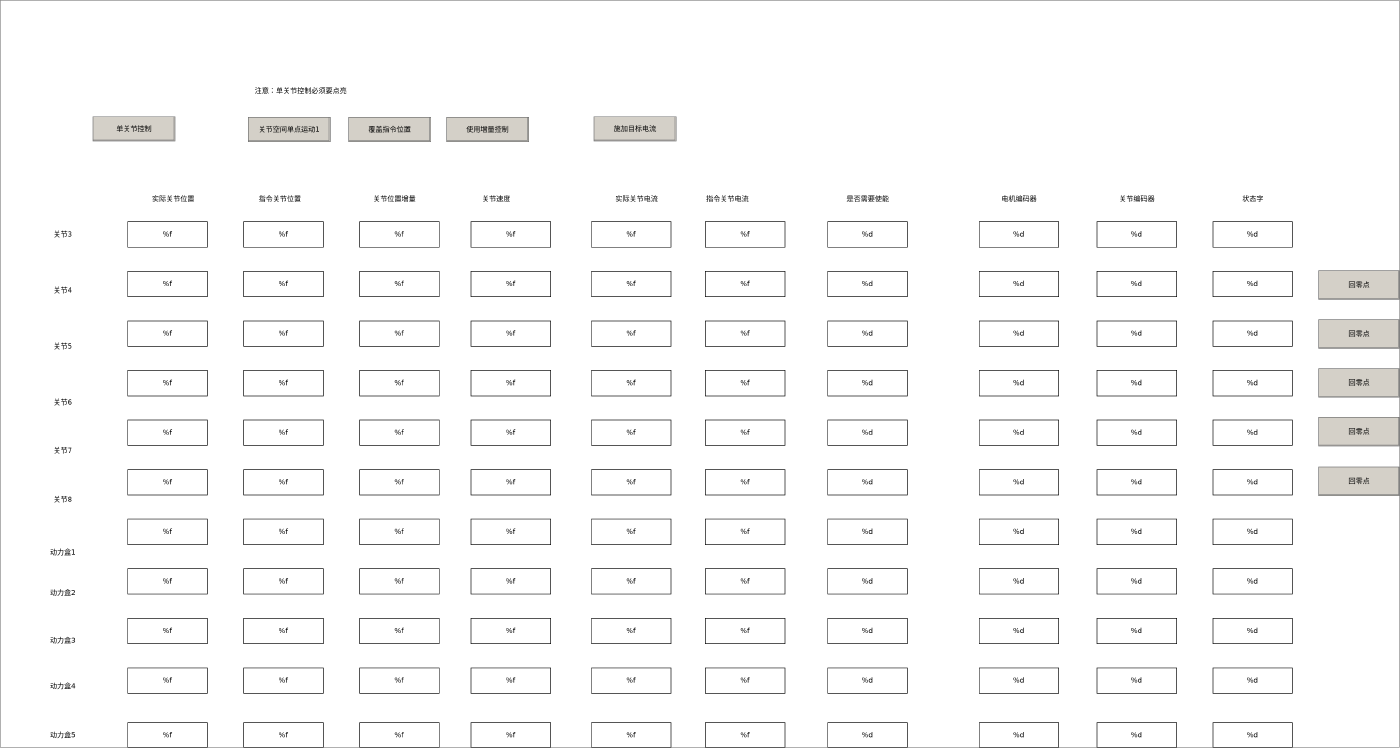
VISUALIZATION motion_a4  // 2174x1162
    Button (385,182 128x38), "关节空间单点运动1", colour toggle: g_motionTest.m_uiArmMode[4,1]
        tap g_motionTest.m_uiArmMode[1,1]
    Label (362,295 145x28), "指令关节位置"
    Label (194,294 150x30), "实际关节位置"
    Label (540,295 145x28), "关节位置增量"
    Label (698,295 145x28), "关节速度"
    Label (916,295 145x28), "实际关节电流"
    Label (1057,295 145x28), "指令关节电流"
    Rectangle (198,575 124x40), "%f", text variable: g_motionTest.m_actJntPos[4][1]
    Label (25,350 145x28), "关节3"
    Label (25,437 145x28), "关节4"
    Label (25,524 145x28), "关节5"
    Label (25,611 145x28), "关节6"
    Label (25,686 145x28), "关节7"
    Label (25,762 145x28), "关节8"
    Label (25,844 145x28), "动力盒1"
    Label (25,907 145x28), "动力盒2"
    Label (25,1128 145x28), "动力盒5"
    Label (25,981 145x28), "动力盒3"
    Label (25,1052 145x28), "动力盒4"
    Rectangle (198,652 124x40), "%f", text variable: g_motionTest.m_actJntPos[4][2]
    Rectangle (198,729 124x40), "%f", text variable: g_motionTest.m_actJntPos[4][3]
    Rectangle (198,806 124x40), "%f", text variable: g_motionTest.m_actJntPos[4][4]
    Rectangle (198,883 124x40), "%f", text variable: g_motionTest.m_actJntPos[4][5]
    Rectangle (198,960 124x40), "%f", text variable: g_motionTest.m_actJntPos[4][6]
    Rectangle (198,1037 124x40), "%f", text variable: g_motionTest.m_actJntPos[4][7]
    Rectangle (198,1122 124x40), "%f", text variable: g_motionTest.m_actJntPos[4][8]
    Rectangle (198,344 124x40), "%f", text variable: g_motionTest.m_actJntPosSetup[4][3]
    Rectangle (198,421 124x40), "%f", text variable: g_motionTest.m_actJntPosSetup[4][4]
    Rectangle (198,498 124x40), "%f", text variable: g_motionTest.m_actJntPosSetup[4][5]
    Rectangle (378,344 124x40), "%f", text variable: g_motionTest.m_targetJntPosSetup[4][3]
        OnMouseClick: write the text variable via Default
    Rectangle (378,421 124x40), "%f", text variable: g_motionTest.m_targetJntPosSetup[4][4]
        OnMouseClick: write the text variable via Default
    Rectangle (378,498 124x40), "%f", text variable: g_motionTest.m_targetJntPosSetup[4][5]
        OnMouseClick: write the text variable via Default
    Rectangle (378,575 124x40), "%f", text variable: g_motionTest.m_targetJntPosN8[4][1]
        OnMouseClick: write the text variable via Default
    Rectangle (378,652 124x40), "%f", text variable: g_motionTest.m_targetJntPosN8[4][2]
        OnMouseClick: write the text variable via Default
    Rectangle (378,729 124x40), "%f", text variable: g_motionTest.m_targetJntPosN8[4][3]
        OnMouseClick: write the text variable via Default
    Rectangle (378,806 124x40), "%f", text variable: g_motionTest.m_targetJntPosN8[4][4]
        OnMouseClick: write the text variable via Default
    Rectangle (378,883 124x40), "%f", text variable: g_motionTest.m_targetJntPosN8[4][5]
        OnMouseClick: write the text variable via Default
    Rectangle (378,960 124x40), "%f", text variable: g_motionTest.m_targetJntPosN8[4][6]
        OnMouseClick: write the text variable via Default
    Rectangle (378,1037 124x40), "%f", text variable: g_motionTest.m_targetJntPosN8[4][7]
        OnMouseClick: write the text variable via Default
    Rectangle (378,1122 124x40), "%f", text variable: g_motionTest.m_targetJntPosN8[4][8]
        OnMouseClick: write the text variable via Default
    Rectangle (558,344 124x40), "%f", text variable: g_motionTest.m_targetJntPosIncSetup[4][3]
        OnMouseClick: write the text variable via Default
    Rectangle (558,421 124x40), "%f", text variable: g_motionTest.m_targetJntPosIncSetup[4][4]
        OnMouseClick: write the text variable via Default
    Rectangle (558,498 124x40), "%f", text variable: g_motionTest.m_targetJntPosIncSetup[4][5]
        OnMouseClick: write the text variable via Default
    Rectangle (558,575 124x40), "%f", text variable: g_motionTest.m_targetJntPosIncN8[4][1]
        OnMouseClick: write the text variable via Default
    Rectangle (558,652 124x40), "%f", text variable: g_motionTest.m_targetJntPosIncN8[4][2]
        OnMouseClick: write the text variable via Default
    Rectangle (558,729 124x40), "%f", text variable: g_motionTest.m_targetJntPosIncN8[4][3]
        OnMouseClick: write the text variable via Default
    Rectangle (558,806 124x40), "%f", text variable: g_motionTest.m_targetJntPosIncN8[4][4]
        OnMouseClick: write the text variable via Default
    Rectangle (558,883 124x40), "%f", text variable: g_motionTest.m_targetJntPosIncN8[4][5]
        OnMouseClick: write the text variable via Default
    Rectangle (558,960 124x40), "%f", text variable: g_motionTest.m_targetJntPosIncN8[4][6]
        OnMouseClick: write the text variable via Default
    Rectangle (558,1037 124x40), "%f", text variable: g_motionTest.m_targetJntPosIncN8[4][7]
        OnMouseClick: write the text variable via Default
    Rectangle (558,1122 124x40), "%f", text variable: g_motionTest.m_targetJntPosIncN8[4][8]
        OnMouseClick: write the text variable via Default
    Rectangle (731,344 124x40), "%f", text variable: g_motionTest.m_targetJntVelSetup[4][3]
        OnMouseClick: write the text variable via Default
    Rectangle (731,421 124x40), "%f", text variable: g_motionTest.m_targetJntVelSetup[4][4]
        OnMouseClick: write the text variable via Default
    Rectangle (731,498 124x40), "%f", text variable: g_motionTest.m_targetJntVelSetup[4][5]
        OnMouseClick: write the text variable via Default
    Rectangle (731,575 124x40), "%f", text variable: g_motionTest.m_targetJntVel[4][1]
        OnMouseClick: write the text variable via Default
    Rectangle (731,652 124x40), "%f", text variable: g_motionTest.m_targetJntVel[4][2]
        OnMouseClick: write the text variable via Default
    Rectangle (731,729 124x40), "%f", text variable: g_motionTest.m_targetJntVel[4][3]
        OnMouseClick: write the text variable via Default
    Rectangle (731,806 124x40), "%f", text variable: g_motionTest.m_targetJntVel[4][4]
        OnMouseClick: write the text variable via Default
    Rectangle (731,883 124x40), "%f", text variable: g_motionTest.m_targetJntVel[4][5]
        OnMouseClick: write the text variable via Default
    Rectangle (731,960 124x40), "%f", text variable: g_motionTest.m_targetJntVel[4][6]
        OnMouseClick: write the text variable via Default
    Rectangle (731,1037 124x40), "%f", text variable: g_motionTest.m_targetJntVel[4][7]
        OnMouseClick: write the text variable via Default
    Rectangle (731,1122 124x40), "%f", text variable: g_motionTest.m_targetJntVel[4][8]
        OnMouseClick: write the text variable via Default
    Rectangle (918,344 124x40), "%f", text variable: g_motionTest.m_actJntCurrentSetup[4][3]
    Rectangle (918,421 124x40), "%f", text variable: g_motionTest.m_actJntCurrentSetup[4][4]
    Rectangle (918,498 124x40), "%f", text variable: g_motionTest.m_actJntCurrentSetup[4][5]
    Rectangle (918,575 124x40), "%f", text variable: g_motionTest.m_actJntCurrent[4][1]
    Rectangle (918,652 124x40), "%f", text variable: g_motionTest.m_actJntCurrent[4][2]
    Rectangle (918,729 124x40), "%f", text variable: g_motionTest.m_actJntCurrent[4][3]
    Rectangle (918,806 124x40), "%f", text variable: g_motionTest.m_actJntCurrent[4][4]
    Rectangle (918,883 124x40), "%f", text variable: g_motionTest.m_actJntCurrent[4][5]
    Rectangle (918,960 124x40), "%f", text variable: g_motionTest.m_actJntCurrent[4][6]
    Rectangle (918,1037 124x40), "%f", text variable: g_motionTest.m_actJntCurrent[4][7]
    Rectangle (918,1122 124x40), "%f", text variable: g_motionTest.m_actJntCurrent[4][8]
    Rectangle (1095,344 124x40), "%f", text variable: g_motionTest.m_targetJntCurrentSetup[4][3]
        OnMouseClick: write the text variable via Default
    Rectangle (1095,421 124x40), "%f", text variable: g_motionTest.m_targetJntCurrentSetup[4][4]
        OnMouseClick: write the text variable via Default
    Rectangle (1095,498 124x40), "%f", text variable: g_motionTest.m_targetJntCurrentSetup[4][5]
        OnMouseClick: write the text variable via Default
    Rectangle (1095,575 124x40), "%f", text variable: g_motionTest.m_targetJntCurrentN8[4][1]
        OnMouseClick: write the text variable via Default
    Rectangle (1095,652 124x40), "%f", text variable: g_motionTest.m_targetJntCurrentN8[4][2]
        OnMouseClick: write the text variable via Default
    Rectangle (1095,729 124x40), "%f", text variable: g_motionTest.m_targetJntCurrentN8[4][3]
        OnMouseClick: write the text variable via Default
    Rectangle (1095,806 124x40), "%f", text variable: g_motionTest.m_targetJntCurrentN8[4][4]
        OnMouseClick: write the text variable via Default
    Rectangle (1095,883 124x40), "%f", text variable: g_motionTest.m_targetJntCurrentN8[4][5]
        OnMouseClick: write the text variable via Default
    Rectangle (1095,960 124x40), "%f", text variable: g_motionTest.m_targetJntCurrentN8[4][6]
        OnMouseClick: write the text variable via Default
    Rectangle (1095,1037 124x40), "%f", text variable: g_motionTest.m_targetJntCurrentN8[4][7]
        OnMouseClick: write the text variable via Default
    Rectangle (1095,1122 124x40), "%f", text variable: g_motionTest.m_targetJntCurrentN8[4][8]
        OnMouseClick: write the text variable via Default
    Button (693,182 128x38), "使用增量控制", colour toggle: g_motionTest.m_singleMotorIncControl[4]
        toggle g_motionTest.m_singleMotorIncControl[4]
    Button (922,181 128x38), "施加目标电流", colour toggle: g_motionTest.m_uiArmMode[4,9]
        toggle g_motionTest.m_uiArmMode[4,9]
    Button (144,181 128x38), "单关节控制", colour toggle: g_motionTest.m_singleMotorControl[4]
        toggle g_motionTest.m_singleMotorControl[4]
    Label (357,126 220x30), "注意：单关节控制必须要点亮"
    Label (1275,294 145x30), "是否需要使能"
    Rectangle (1285,344 124x40), "%d", text variable: g_motionTest.m_jntEnableSetup[4][3]
        OnMouseClick: write the text variable via Default
    Rectangle (1285,421 124x40), "%d", text variable: g_motionTest.m_jntEnableSetup[4][4]
        OnMouseClick: write the text variable via Default
    Rectangle (1285,498 124x40), "%d", text variable: g_motionTest.m_jntEnableSetup[4][5]
        OnMouseClick: write the text variable via Default
    Rectangle (1285,575 124x40), "%d", text variable: g_motionTest.m_jntEnable[4][1]
        OnMouseClick: write the text variable via Default
    Rectangle (1285,652 124x40), "%d", text variable: g_motionTest.m_jntEnable[4][2]
        OnMouseClick: write the text variable via Default
    Label (1510,295 145x28), "电机编码器"
    Label (1693,295 145x28), "关节编码器"
    Label (1873,295 145x28), "状态字"
    Rectangle (1520,344 124x40), "%d", text variable: g_systemInfo.m_setupJntInfo[4,3].m_motorInput.m_motorEncoder
    Rectangle (1520,421 124x40), "%d", text variable: g_systemInfo.m_setupJntInfo[4,4].m_motorInput.m_motorEncoder
    Rectangle (1520,498 124x40), "%d", text variable: g_systemInfo.m_setupJntInfo[4,5].m_motorInput.m_motorEncoder
    Rectangle (1520,575 124x40), "%d", text variable: g_systemInfo.m_slaveJntInfo[4,1].m_motorInput.m_motorEncoder
    Rectangle (1520,652 124x40), "%d", text variable: g_systemInfo.m_slaveJntInfo[4,2].m_motorInput.m_motorEncoder
    Rectangle (1703,344 124x40), "%d", text variable: g_systemInfo.m_setupJntInfo[4,3].m_motorInput.m_linkEncoder
    Rectangle (1703,421 124x40), "%d", text variable: g_systemInfo.m_setupJntInfo[4,4].m_motorInput.m_linkEncoder
    Rectangle (1703,498 124x40), "%d", text variable: g_systemInfo.m_setupJntInfo[4,5].m_motorInput.m_linkEncoder
    Rectangle (1703,575 124x40), "%d", text variable: g_systemInfo.m_slaveJntInfo[4,1].m_motorInput.m_linkEncoder
    Rectangle (1703,652 124x40), "%d", text variable: g_systemInfo.m_slaveJntInfo[4,2].m_motorInput.m_linkEncoder
    Rectangle (1883,344 124x40), "%d", text variable: g_systemInfo.m_setupJntInfo[4,3].m_motorInput.m_statusWord
    Rectangle (1883,421 124x40), "%d", text variable: g_systemInfo.m_setupJntInfo[4,4].m_motorInput.m_statusWord
    Rectangle (1883,498 124x40), "%d", text variable: g_systemInfo.m_setupJntInfo[4,5].m_motorInput.m_statusWord
    Rectangle (1883,575 124x40), "%d", text variable: g_systemInfo.m_slaveJntInfo[4,1].m_motorInput.m_statusWord
    Rectangle (1883,652 124x40), "%d", text variable: g_systemInfo.m_slaveJntInfo[4,2].m_motorInput.m_statusWord
    Rectangle (1520,729 124x40), "%d", text variable: g_systemInfo.m_slaveJntInfo[4,3].m_motorInput.m_motorEncoder
    Rectangle (1520,806 124x40), "%d", text variable: g_systemInfo.m_slaveJntInfo[4,4].m_motorInput.m_motorEncoder
    Rectangle (1520,883 124x40), "%d", text variable: g_systemInfo.m_slaveJntInfo[4,5].m_motorInput.m_motorEncoder
    Rectangle (1520,960 124x40), "%d", text variable: g_systemInfo.m_slaveJntInfo[4,6].m_motorInput.m_motorEncoder
    Rectangle (1520,1037 124x40), "%d", text variable: g_systemInfo.m_slaveJntInfo[4,7].m_motorInput.m_motorEncoder
    Rectangle (1520,1122 124x40), "%d", text variable: g_systemInfo.m_slaveJntInfo[4,8].m_motorInput.m_motorEncoder
    Rectangle (1703,729 124x40), "%d", text variable: g_systemInfo.m_slaveJntInfo[4,3].m_motorInput.m_linkEncoder
    Rectangle (1703,806 124x40), "%d", text variable: g_systemInfo.m_slaveJntInfo[4,4].m_motorInput.m_linkEncoder
    Rectangle (1703,883 124x40), "%d", text variable: g_systemInfo.m_slaveJntInfo[4,5].m_motorInput.m_linkEncoder
    Rectangle (1703,960 124x40), "%d", text variable: g_systemInfo.m_slaveJntInfo[4,6].m_motorInput.m_linkEncoder
    Rectangle (1703,1037 124x40), "%d", text variable: g_systemInfo.m_slaveJntInfo[4,7].m_motorInput.m_linkEncoder
    Rectangle (1703,1122 124x40), "%d", text variable: g_systemInfo.m_slaveJntInfo[4,8].m_motorInput.m_linkEncoder
    Rectangle (1883,729 124x40), "%d", text variable: g_systemInfo.m_slaveJntInfo[4,3].m_motorInput.m_statusWord
    Rectangle (1883,806 124x40), "%d", text variable: g_systemInfo.m_slaveJntInfo[4,4].m_motorInput.m_statusWord
    Rectangle (1883,883 124x40), "%d", text variable: g_systemInfo.m_slaveJntInfo[4,5].m_motorInput.m_statusWord
    Rectangle (1883,960 124x40), "%d", text variable: g_systemInfo.m_slaveJntInfo[4,6].m_motorInput.m_statusWord
    Rectangle (1883,1037 124x40), "%d", text variable: g_systemInfo.m_slaveJntInfo[4,7].m_motorInput.m_statusWord
    Rectangle (1883,1122 124x40), "%d", text variable: g_systemInfo.m_slaveJntInfo[4,8].m_motorInput.m_statusWord
    Rectangle (1285,729 124x40), "%d", text variable: g_motionTest.m_jntEnable[4][3]
        OnMouseClick: write the text variable via Default
    Rectangle (1285,806 124x40), "%d", text variable: g_motionTest.m_jntEnable[4][4]
        OnMouseClick: write the text variable via Default
    Rectangle (1285,883 124x40), "%d", text variable: g_motionTest.m_jntEnable[4][5]
        OnMouseClick: write the text variable via Default
    Rectangle (1285,960 124x40), "%d", text variable: g_motionTest.m_jntEnable[4][6]
        OnMouseClick: write the text variable via Default
    Rectangle (1285,1037 124x40), "%d", text variable: g_motionTest.m_jntEnable[4][7]
        OnMouseClick: write the text variable via Default
    Rectangle (1285,1122 124x40), "%d", text variable: g_motionTest.m_jntEnable[4][8]
        OnMouseClick: write the text variable via Default
    Button (541,182 128x38), "覆盖指令位置", colour toggle: g_motionTest.m_coverCmdPos[4]
        tap g_motionTest.m_coverCmdPos[4]
    Button (2047,420 127x45), "回零点", colour toggle: g_motionTest.m_goHomeSetup[4][4]
        tap g_motionTest.m_goHomeSetup[4][4]
    Button (2047,496 127x45), "回零点", colour toggle: g_motionTest.m_goHomeSetup[4][5]
        tap g_motionTest.m_goHomeSetup[4][5]
    Button (2047,572 127x45), "回零点", colour toggle: g_motionTest.m_goHome[4][1]
        tap g_motionTest.m_goHome[4][1]
    Button (2047,648 127x45), "回零点", colour toggle: g_motionTest.m_goHome[4][2]
        tap g_motionTest.m_goHome[4][2]
    Button (2047,725 127x45), "回零点", colour toggle: g_motionTest.m_goHome[4][3]
        tap g_motionTest.m_goHome[4][3]
END_VISUALIZATION

(* stored: Version 1.1.0.1, ProductVersion 3.1.4024.11
   Visu motion_a4: Id {291468c6-ac84-4b8c-ac21-6db673ee89db} *)
